// TwinCAT 3 PLC project SPS
// ProgramVersion: 3.1.4024.0
// libraries:
//   Tc2_MC2, * (Beckhoff Automation GmbH)
//   Tc2_Standard, * (Beckhoff Automation GmbH)
//   Tc2_System, * (Beckhoff Automation GmbH)
//   Tc3_Module, * (Beckhoff Automation GmbH)
// project tree:
//   DUTs/ eBetriebszustand.TcDUT
//   GVLs/ GVL_PosKinematic.TcGVL, IFC_HW.TcGVL (not stored)
//   / PlcTask.TcTTO
//   POUs/ FB_Abfuellmodul.TcPOU, FB_Ampel.TcPOU, FB_Blinklicht.TcPOU, FB_Dispenser.TcPOU, FB_EZylinder.TcPOU, FB_Manipulatormodul.TcPOU, FB_Maschinentuer.TcPOU, FB_TEST.TcPOU, FUN_SCALE.TcPOU, MAIN.TcPOU, FB_Vereinzelung.TcPOU
//   POUs/Manipulator/ FB_MANACHSE.TcPOU, FB_Robotsteuerung.TcPOU
//   POUs/Transport/ FB_Foerderband.TcPOU, FB_Transport.TcPOU, FB_TransportA.TcPOU, FB_TransportE.TcPOU, FB_TransportLogik.TcPOU
// real-time tasks:
//   TASK PlcTask: cycle T#10ms, priority 20, ADS port 350
// motion (NC):
//   TASK NC-Task 1 SAF: cycle T#2ms, priority 4, ADS port 501
//   TASK NC-Task 1 SVB: cycle T#10ms, priority 8, ADS port 511
//   AXIS Conveyer (id 1)
//     Dynamic: AccelerationMaximum=700, DecelerationMaximum=700, Acceleration=400, Deceleration=400, Jerk=6000
//     Velo: Maximum=50
//     OtherSettings: AllowMotionCmdToSlave=true
//     encoder EncType=1
//     drive DrvType=5
//       Analog: VeloReferenz=50, TorqueSetpointScale=10, ScaleFactorActTorque=0.1
//       TimeComp: TaskDelayCycles=1
//     controller CtrType=1
//       CtrPara: PriorControlFactor=1
//         Observer: BandWidth=20
//   AXIS Dispenser1 (id 2)
//     Dynamic: AccelerationMaximum=700, DecelerationMaximum=700, Acceleration=400, Deceleration=400, Jerk=6000
//     Velo: Maximum=50
//     OtherSettings: AllowMotionCmdToSlave=true
//     encoder EncType=1
//     drive DrvType=5
//       Analog: VeloReferenz=50, TorqueSetpointScale=10, ScaleFactorActTorque=0.1
//       TimeComp: TaskDelayCycles=1
//     controller CtrType=1
//       CtrPara: PriorControlFactor=1
//         Observer: BandWidth=20
//   AXIS Dispenser2 (id 3)
//     Dynamic: AccelerationMaximum=700, DecelerationMaximum=700, Acceleration=400, Deceleration=400, Jerk=6000
//     Velo: Maximum=50
//     OtherSettings: AllowMotionCmdToSlave=true
//     encoder EncType=1
//     drive DrvType=5
//       Analog: VeloReferenz=50, TorqueSetpointScale=10, ScaleFactorActTorque=0.1
//       TimeComp: TaskDelayCycles=1
//     controller CtrType=1
//       CtrPara: PriorControlFactor=1
//         Observer: BandWidth=20
//   AXIS Dispenser3 (id 4)
//     Dynamic: AccelerationMaximum=700, DecelerationMaximum=700, Acceleration=400, Deceleration=400, Jerk=6000
//     Velo: Maximum=50
//     OtherSettings: AllowMotionCmdToSlave=true
//     encoder EncType=1
//     drive DrvType=5
//       Analog: VeloReferenz=50, TorqueSetpointScale=10, ScaleFactorActTorque=0.1
//       TimeComp: TaskDelayCycles=1
//     controller CtrType=1
//       CtrPara: PriorControlFactor=1
//         Observer: BandWidth=20
//   AXIS ManAchseX (id 5)
//     Dynamic: AccelerationMaximum=700, DecelerationMaximum=700, Acceleration=400, Deceleration=400, Jerk=6000
//     Velo: Maximum=30
//     OtherSettings: AllowMotionCmdToSlave=true
//     encoder EncType=1
//       EncPara: ScaleFactorNumerator=0.0025
//         Inc: RefSearchInverse=true, RefSyncInverse=false
//     drive DrvType=5
//       Analog: VeloReferenz=30, TorqueSetpointScale=10, ScaleFactorActTorque=0.1
//       TimeComp: TaskDelayCycles=1
//     controller CtrType=1
//       CtrPara: PriorControlFactor=1
//         Observer: BandWidth=20
//   AXIS ManAchseY (id 6)
//     Dynamic: AccelerationMaximum=700, DecelerationMaximum=700, Acceleration=400, Deceleration=400, Jerk=6000
//     Velo: Maximum=30
//     OtherSettings: AllowMotionCmdToSlave=true
//     encoder EncType=1
//       EncPara: ScaleFactorNumerator=0.0025
//         Inc: RefSearchInverse=true, RefSyncInverse=false
//     drive DrvType=5
//       Analog: VeloReferenz=30, TorqueSetpointScale=10, ScaleFactorActTorque=0.1
//       TimeComp: TaskDelayCycles=1
//     controller CtrType=1
//       CtrPara: PriorControlFactor=1
//         Observer: BandWidth=20
//   AXIS ManAchseZ (id 7)
//     Dynamic: AccelerationMaximum=700, DecelerationMaximum=700, Acceleration=400, Deceleration=400, Jerk=6000
//     Velo: Maximum=30
//     OtherSettings: AllowMotionCmdToSlave=true
//     encoder EncType=1
//       EncPara: ScaleFactorNumerator=0.0025
//         Inc: RefSearchInverse=true, RefSyncInverse=false
//     drive DrvType=5
//       Analog: VeloReferenz=30, TorqueSetpointScale=10, ScaleFactorActTorque=0.1
//       TimeComp: TaskDelayCycles=1
//     controller CtrType=1
//       CtrPara: PriorControlFactor=1
//         Observer: BandWidth=20
//   AXIS ManAchseG (id 8)
//     Dynamic: AccelerationMaximum=700, DecelerationMaximum=700, Acceleration=400, Deceleration=400, Jerk=6000
//     Velo: Maximum=30
//     OtherSettings: AllowMotionCmdToSlave=true
//     encoder EncType=1
//       EncPara: ScaleFactorNumerator=0.0025
//     drive DrvType=5
//       Analog: VeloReferenz=30, TorqueSetpointScale=10, ScaleFactorActTorque=0.1
//     controller CtrType=1
//       CtrPara: PriorControlFactor=1
//         Observer: BandWidth=20
// variable links:
//   SPS/SPS Instance <-> NC-Task 1 SAF/Axes/Conveyer
//     PlcTask Inputs/IFC_HW.ax_BandMotor.NcToPlc <-> Outputs/ToPlc
//     PlcTask Outputs/IFC_HW.ax_BandMotor.PlcToNc <-> Inputs/FromPlc
//   SPS/SPS Instance <-> NC-Task 1 SAF/Axes/Dispenser1
//     PlcTask Inputs/IFC_HW.ax_Extruder1.NcToPlc <-> Outputs/ToPlc
//     PlcTask Outputs/IFC_HW.ax_Extruder1.PlcToNc <-> Inputs/FromPlc
//   SPS/SPS Instance <-> NC-Task 1 SAF/Axes/Dispenser2
//     PlcTask Inputs/IFC_HW.ax_Extruder2.NcToPlc <-> Outputs/ToPlc
//     PlcTask Outputs/IFC_HW.ax_Extruder2.PlcToNc <-> Inputs/FromPlc
//   SPS/SPS Instance <-> NC-Task 1 SAF/Axes/Dispenser3
//     PlcTask Inputs/IFC_HW.ax_Extruder3.NcToPlc <-> Outputs/ToPlc
//     PlcTask Outputs/IFC_HW.ax_Extruder3.PlcToNc <-> Inputs/FromPlc
//   SPS/SPS Instance <-> NC-Task 1 SAF/Axes/ManAchseG
//     PlcTask Inputs/IFC_HW.ax_ManG.NcToPlc <-> Outputs/ToPlc
//     PlcTask Outputs/IFC_HW.ax_ManG.PlcToNc <-> Inputs/FromPlc
//   SPS/SPS Instance <-> NC-Task 1 SAF/Axes/ManAchseX
//     PlcTask Inputs/IFC_HW.ax_ManX.NcToPlc <-> Outputs/ToPlc
//     PlcTask Outputs/IFC_HW.ax_ManX.PlcToNc <-> Inputs/FromPlc
//   SPS/SPS Instance <-> NC-Task 1 SAF/Axes/ManAchseY
//     PlcTask Inputs/IFC_HW.ax_ManY.NcToPlc <-> Outputs/ToPlc
//     PlcTask Outputs/IFC_HW.ax_ManY.PlcToNc <-> Inputs/FromPlc
//   SPS/SPS Instance <-> NC-Task 1 SAF/Axes/ManAchseZ
//     PlcTask Inputs/IFC_HW.ax_ManZ.NcToPlc <-> Outputs/ToPlc
//     PlcTask Outputs/IFC_HW.ax_ManZ.PlcToNc <-> Inputs/FromPlc

CONFIGURATION SPS
    RESOURCE PLC ON TwinCAT3
        TASK PlcTask(INTERVAL := T#10ms, PRIORITY := 20);
        PROGRAM MAIN WITH PlcTask : MAIN;
    END_RESOURCE
END_CONFIGURATION

// ---- DUTs/eBetriebszustand.TcDUT
{attribute 'qualified_only'}
{attribute 'strict'}
TYPE eBetriebszustand :
(
	off, //nicht Betriebsbereit 
	error, //Fehlerbehafteter Stop(Sicherheitssteuerung)
	setup, //Wartung 
	warning, // Nicht fehlerbehafteter geplanter Stop 
	init, //Herstellung Betriebsbereitschaft 
	ready, //betriebsbereit 
	production, //Im Betrieb
	done, //Betrieb abgschlossen
	stop //geplanter Stillstand 
);
END_TYPE

// ---- GVLs/GVL_PosKinematic.TcGVL
{attribute 'qualified_only'}
VAR_GLOBAL
	// Home position
	pXhome : REAL := 29;
	pYhome : REAL := 145.5;
	pZhome : REAL := 45;
	
	// Conveyor position
	pXconv : REAL := 29;
	pYconv : REAL := 145.5;
	pZconv : REAL := 130;
	
	//Scale position
	pXscale : REAL := 36;
	pYscale : REAL := 7.5;
	pZscale : REAL := 131.5;
	
	// Heating position
	pXheat : REAL := 218.5;
	pYheat : REAL := 7;
	pZheat : REAL := 159;
	
	// Storage position
	pX1stor : REAL := 107;
	pX2stor : REAL := 158.7;
	pX3stor : REAL := 209.3;
	pX4stor : REAL := 260.3;
	pYstor : REAL := 139;
	pZstor : REAL := 120;
	
	// Z offset height
	pZoff : REAL := 45;
END_VAR

// ---- POUs/MAIN.TcPOU
PROGRAM MAIN
VAR
	fbBlinklicht : FB_Blinklicht;
	fbVereinzelung : FB_Vereinzelung;
	fbezylinder1 : FB_EZylinder;
	fbezylinder2 : FB_EZylinder;
	fbAmpel : FB_Ampel;
	fbTransport : FB_Transport;
	fbDispenser : FB_Dispenser;
	fbAbfuellmodul : FB_Abfuellmodul;
	fbManAchseX : FB_ManAchse;
	fbManAchseY : FB_ManAchse;
	fbManAchseZ : FB_ManAchse;
	fbManAchseG : FB_ManAchse;
	fbRobotsteuerung : FB_Robotsteuerung;
	fbManipulatormodul : FB_Manipulatormodul;
	ix : UINT;
	ry : REAL;
	ax : Axis_Ref;
END_VAR

ry := FUN_SCALE(TO_REAL(ix),4096,0,350,0);

	
fbAbfuellmodul(
	bEnable:= IFC_HW.bEnable, 
	bExecute:= IFC_HW.bExecute, 
	nstation:= , 
	bEinzelSens1:= IFC_HW.bEinzelSens1, 
	bEinzelSens2:= IFC_HW.bEinzelSens2, 
	bEinzelSens3:= IFC_HW.bEinzelSens3, 
	bEinzelSens4:= IFC_HW.bBandSens1, 
	bBandSens1:= IFC_HW.bBandSens1, 
	bBandSens2:= IFC_HW.bBandSens2, 
	bBandSens3:= IFC_HW.bBandSens3, 
	bBandSens4:= IFC_HW.bBandSens4, 
	bstopper1=> IFC_HW.bBandHub1, 
	bstopper2=> IFC_HW.bBandHub2, 
	bstopper3=>IFC_HW.bBandHub3, 
	estate=> , 
	bgate1=> fbeZylinder1.bgate, 
	bgate2=> fbeZylinder2.bgate, 
	axTransport:= IFC_HW.ax_BandMotor, 
	axDisp1:= IFC_HW.ax_Extruder1, 
	axDisp2:= IFC_HW.ax_Extruder2, 
	axDisp3:= IFC_HW.ax_Extruder3);
	
	fbezylinder1(bgate:= , berror:= , bR1=>IFC_HW.bR1AKT1 , bR2=>IFC_HW.br2AKT1 );
	
	fbezylinder2(bgate:= , berror:= , bR1=>IFC_HW.bR1AKT2 , bR2=> IFC_HW.bR2AKT2);
	
	
	fbAmpel(estate:= fbAbfuellmodul.estate, bAmpelgruen=>IFC_HW.bAmpelGrun , bAmpelrot=>IFC_HW.bAmpelRot , bAmpelgelb=>IFC_HW.bAmpelGelb );

fbManipulatormodul(
	bEnable:= IFC_Hw.bEnable, 
	bExecute:= IFC_Hw.bExecute, 
	pXhome:= GVL_PosKinematic.pXhome, 
	pYhome:= GVL_PosKinematic.pYhome, 
	pZhome:= GVL_PosKinematic.pZhome, 
	pXconv:= GVL_PosKinematic.pXconv, 
	pYconv:= GVL_PosKinematic.pYconv, 
	pZconv:= GVL_PosKinematic.pZconv, 
	pXscale:= GVL_PosKinematic.pXscale, 
	pYscale:= GVL_PosKinematic.pYscale, 
	pZscale:= GVL_PosKinematic.pZscale, 
	pXheat:= GVL_PosKinematic.pXheat, 
	pYheat:= GVL_PosKinematic.pYheat, 
	pZheat:= GVL_PosKinematic.pZheat, 
	pX1stor:= GVL_PosKinematic.pX1stor, 
	pX2stor:= GVL_PosKinematic.pX2stor, 
	pX3stor:= GVL_PosKinematic.pX3stor, 
	pX4stor:= GVL_PosKinematic.pX4stor, 
	pYstor:= GVL_PosKinematic.pYstor, 
	pZstor:= GVL_PosKinematic.pZstor, 
	estateE:= fbAbfuellmodul.estate, 
	bxEndschalter:= IFC_HW.bManEndXmin, 
	byEndschalter:= IFC_HW.bManEndYmin, 
	bzEndschalter:= IFC_HW.bManEndZmin, 
	bGEndschalter:= IFC_HW.bManEndGmin, 
	estate=> , 
	ax_ManX:= IFC_HW.ax_ManX, 
	ax_ManY:= IFC_HW.ax_ManY, 
	ax_ManZ:= IFC_HW.ax_ManZ, 
	ax_ManG:= IFC_HW.ax_ManG);

(*
fbRobotsteuerung(
	bEnable:= IFC_Hw.bEnable, 
	bExecute:= IFC_Hw.bExecute, 
	bxposition:= GVL_PosKinematic.pXconv, 
	byposition:= GVL_PosKinematic.pYconv, 
	bzposition:= GVL_PosKinematic.pZconv, 
	bxEndschalter:= IFC_HW.bManEndXmin, 
	byEndschalter:= IFC_HW.bManEndYmin, 
	bzEndschalter:= IFC_HW.bManEndZmin, 
	bGEndschalter:= IFC_HW.bManEndGmin, 
	estateE:= fbAbfuellmodul.estate, 
	estate=> , 
	movedone=> , 
	ax_ManX:= IFC_HW.ax_ManX, 
	ax_ManY:= IFC_HW.ax_ManY, 
	ax_ManZ:= IFC_HW.ax_ManZ, 
	ax_ManG:= IFC_HW.ax_ManG);

fbManAchseX(
	benable:= IFC_Hw.bEnable, 
	bexecute:= IFC_Hw.bExecute, 
	bEndschalter:= IFC_HW.bManEndXmin, 
	rPosition:= GVL_PosKinematic.pXconv, 
	rVel:= 30, 
	estate=> , 
	ax:= IFC_HW.ax_ManX);
	
fbManAchseY(
	benable:= IFC_Hw.bEnable, 
	bexecute:= IFC_Hw.bExecute, 
	bEndschalter:= IFC_HW.bManEndYmin, 
	rPosition:= GVL_PosKinematic.pYconv, 
	rVel:= 30, 
	estate=> , 
	ax:= IFC_HW.ax_ManY); 

fbManAchseZ(
	benable:= IFC_Hw.bEnable, 
	bexecute:= IFC_Hw.bExecute, 
	bEndschalter:= IFC_HW.bManEndZmin, 
	rPosition:= GVL_PosKinematic.pZconv, 
	rVel:= 30, 
	estate=> , 
	ax:= IFC_HW.ax_ManZ); 	

fbManAchseG(
	benable:= IFC_Hw.bEnable, 
	bexecute:= IFC_Hw.bExecute, 
	bEndschalter:= IFC_HW.bManEndGmin, 
	rPosition:= 2, 
	rVel:= 30, 
	estate=> , 
	ax:= IFC_HW.ax_ManG);
*)

END_PROGRAM

// ---- POUs/FB_Blinklicht.TcPOU
FUNCTION_BLOCK FB_Blinklicht
VAR_INPUT
	bStartStop	: BOOL;
	tPeriode	: TIME := T#1.5S;
END_VAR
VAR_OUTPUT
	bBlink	:BOOL;
END_VAR
VAR
	fbTon	:Ton;
	fbRtrig	:R_Trig;
	bEinAus	:BOOL;
END_VAR

fbRtrig(CLK:= bStartStop , Q=> );

IF fbRtrig.Q THEN
	bEinAus := NOT bEinAus;
END_IF

//fbTon.IN := bBlink AND NOT fbTon.Q;
//fbTon.PT := T#1S;

fbTon(IN:=bEinAus AND NOT fbTon.Q , PT:=T#1.5S , Q=> , ET=> );


IF fbTon.ET <= fbTon.PT/2 THEN 
	bBlink := FALSE;
ELSIF fbTon.ET > fbTon.PT/2 THEN
	bBlink := TRUE;
END_IF

END_FUNCTION_BLOCK

// ---- POUs/FB_Vereinzelung.TcPOU
FUNCTION_BLOCK FB_Vereinzelung 
VAR_INPUT
	//Steuervariablen
	benable : BOOL;
	bexecute : BOOL;
	// Hardware Eingänge
	bsensor1 : BOOL; //Flasche in der Kammer 
	bsensor2 : BOOL; //Flasche inm Rohr 
	bsensor3 : BOOL; //Flasche auf Kopf
	bsensor4 : BOOL; //Flasche am Förderband
	
END_VAR
VAR_OUTPUT
	//Hardwareausgänge 
	bgate1 : BOOL;
	bgate2 : BOOL;
	//Steuervariable 
	estate : eBetriebszustand;
END_VAR
VAR
	nstate : INT := 100;
	fbTon : Ton;
END_VAR

fbTon(IN:= , PT:=T#1S , Q=> , ET=> );

CASE nstate OF 
	100:
	eState :=eBetriebszustand.off;
	
	IF bsensor1 AND benable THEN 
		nstate := 21;//Ready
	ELSIF benable THEN
		nstate := 0; //Init		
	END_IF
	
	0: // Kammer ist leer 
	estate := eBetriebszustand.init;
	bgate1 := FALSE;
	bgate2 := FALSE;
	
	IF bsensor2 AND NOT bsensor3 THEN
		nstate := 1; //Schleuße Oben öffnen
	END_IF
	
	1: // Schleuße oben öffnen
	estate := eBetriebszustand.init;
	bgate1 := TRUE;
	bgate2 := FALSE;
	
	IF bsensor1 THEN
		nstate := 2; //Schleuße oben schließen
	END_IF
	
	2: //Schleuße oben schließen
	estate := eBetriebszustand.init;
	bgate1 := FALSE;
	bgate2 := FALSE;
	fbTon.In := TRUE;
	
	IF fbTon.Q THEN
		nstate := 21; //ready
		fbTon.IN := FALSE;
	END_IF
	
	21: //ready
	estate:= eBetriebszustand.ready;
	bgate1:= FALSE;
	bgate2:= FALSE;
	
	
	IF bexecute THEN
		nstate := 3; //Schleuße unten öffnen
	END_IF
	
	3: //Schleuße unten öffnen
	estate:= eBetriebszustand.production;
	bgate1:= FALSE;
	bgate2:= TRUE;
	
	IF bsensor4 THEN
		nstate := 4; //Schleuße unten schließen
	END_IF
	
	4: //Schleuße unten schließen
	estate:= eBetriebszustand.production;
	bgate1:= FALSE;
	bgate2:= FALSE;
	fbTon.IN:= TRUE;
	
	IF fbTon.Q THEN
		nstate := 41; //done
		fbTon.IN := FALSE;
	END_IF	
	
	41: //Done
	estate:= eBetriebszustand.done;
	bgate1:= FALSE;
	bgate2:= FALSE;
	
	IF NOT bexecute THEN
		nstate:= 0; //Kammer leer
	END_IF
	
END_CASE

END_FUNCTION_BLOCK

// ---- POUs/FB_EZylinder.TcPOU
FUNCTION_BLOCK FB_EZylinder
VAR_INPUT
	bgate : BOOL;
	berror : BOOL;
END_VAR
VAR_OUTPUT
	bR1 : BOOL;
	bR2 : BOOL;
END_VAR
VAR
END_VAR


bR1 := bgate;
bR2 := NOT bgate;

IF berror THEN
	bR1 := FALSE;
	bR2 := FALSE;
	
END_IF

END_FUNCTION_BLOCK

// ---- POUs/FB_Ampel.TcPOU
FUNCTION_BLOCK FB_Ampel
VAR_INPUT
	estate : eBetriebszustand;
END_VAR
VAR_OUTPUT
	bAmpelgruen : BOOL;
	bAmpelrot : BOOL;
	bAmpelgelb : BOOL;
END_VAR
VAR
	Ampel_blinken : FB_Blinklicht;
END_VAR

//Die Ampel leuchtet je nach Betriebszustand in unterschiedlichen Farben, um diesen anzuzeigen
CASE estate OF
	
	eBetriebszustand.off:
	bAmpelgruen := FALSE;
	bAmpelrot := TRUE;
	bAmpelgelb := FALSE;	
	
	eBetriebszustand.init:
	bAmpelrot := FALSE;
	bAmpelgelb := FALSE;
	Ampel_blinken(bStartStop:=TRUE , tPeriode:= , bBlink=>bAmpelgruen );
	
	eBetriebszustand.ready:
	bAmpelrot := FALSE;
	Ampel_blinken(bStartStop:=TRUE , tPeriode:= , bBlink=>bAmpelgelb );
	bAmpelgruen := NOT bAmpelgelb;
	//gruen_blinken(bStartStop:=True , tPeriode:= , bBlink=>bAmpelgruen );
	
	eBetriebszustand.production:
	bAmpelrot := FALSE;
	bAmpelgelb := FALSE;
	bAmpelgruen := TRUE;
	
	eBetriebszustand.done:
	bAmpelgruen := TRUE;
	bAmpelrot := FALSE;
	bAmpelgelb := TRUE;	
	
END_CASE

END_FUNCTION_BLOCK

// ---- POUs/Transport/FB_Transport.TcPOU
FUNCTION_BLOCK FB_Transport
VAR_INPUT
	bEnable : BOOL;
	bExecute : BOOL;
	nstation : INT;
	//Hardware Eingänge
	bSens1 : BOOL;
	bSens2 : BOOL;
	bSens3 : BOOL;
	bSens4 : BOOL;
END_VAR
VAR_OUTPUT
	eState : eBetriebszustand;
	bstopper1 : BOOL;
	bstopper2 : BOOL;
	bstopper3 : BOOL;
	
END_VAR
VAR
	fbTransportE : FB_TransportE;
	fbTransportLogik : FB_TransportLogik;
	fbTransportBand : FB_Foerderband;
	fbTransportA : FB_TransportA;
END_VAR
VAR_IN_OUT
	//Achsenreferenz
	ax : Axis_Ref;
END_VAR

fbTransportE(
	bSens1:= bSens1, 
	bSens2:= bSens2, 
	bSens3:= bSens3, 
	bSens4:= bSens4, 
	bStation1=> , 
	bStation2=> , 
	bStation3=> , 
	bStation4=> );
	
	
fbTransportLogik(
	bEnable:= bEnable, 
	bExecute:= bExecute, 
	eStateE:= fbTransportBand.estate, 
	nStation:= nstation, 
	bStation1:= fbTransportE.bStation1, 
	bStation2:= fbTransportE.bStation2, 
	bStation3:= fbTransportE.bStation3, 
	bStation4:= fbTransportE.bStation4, 
	bEnableA=> , 
	bExecuteA=> , 
	bStopA=> , 
	eStateA=> estate, 
	bStop1=> , 
	bStop2=> , 
	bStop3=> );	
	
fbTransportBand(
	benable:= fbTransportLogik.bEnableA, 
	bexecute:= fbTransportLogik.bExecuteA, 
	bhalt:= fbTransportLogik.bStopA, 
	rVel:= 30, 
	eDirection:= MC_Positive_Direction, 
	estate=> , 
	ax:= ax);

fbTransportA(
	bstop1:= fbTransportLogik.bStop1, 
	bstop2:= fbTransportLogik.bStop2, 
	bstop3:= fbTransportLogik.bStop3, 
	bstopper1=> bStopper1, 
	bstopper2=> bStopper2, 
	bstopper3=> bStopper3);

END_FUNCTION_BLOCK

// ---- POUs/Transport/FB_TransportE.TcPOU
FUNCTION_BLOCK FB_TransportE
VAR_INPUT
	bSens1 : BOOL;
	bSens2 : BOOL;
	bSens3 : BOOL;
	bSens4 : BOOL;
END_VAR
VAR_OUTPUT
	bStation1 : BOOL;
	bStation2 : BOOL;
	bStation3 : BOOL;
	bStation4 : BOOL;
END_VAR
VAR
END_VAR

bStation1 := bSens1;
bStation2 := bSens2;
bStation3 := bSens3;
bStation4 := bSens4;

END_FUNCTION_BLOCK

// ---- POUs/Transport/FB_TransportLogik.TcPOU
FUNCTION_BLOCK FB_TransportLogik
VAR_INPUT
	bEnable : BOOL;
    bExecute : BOOL;
    eStateE : eBetriebszustand;
    nStation : INT := 0;

    // Logiksignale -> Hardware Signale
    bStation1 : BOOL;
    bStation2 : BOOL;
    bStation3 : BOOL;
    bStation4 : BOOL;
END_VAR
VAR_OUTPUT
	bEnableA : BOOL;
    bExecuteA : BOOL;
    eStateA : eBetriebszustand;
	bStopA : BOOL;
    //Hardware Signale -> Logik
    bStop1 : BOOL;
    bStop2 : BOOL;
    bStop3 : BOOL;
END_VAR
VAR
	nstate : INT;
END_VAR

CASE nstate OF 
	0: //Off
	bEnableA := FALSE;
	bExecuteA := FALSE;
	bStopA := FALSE;
	bStop1 := FALSE;
	bStop2 := FALSE;
	bStop3 := FALSE;
	eStateA    := eBetriebszustand.off;
	
	IF bEnable THEN
		nstate := 1; //Init
	END_IF
	
	1: //Init
	bEnableA := TRUE;
	bExecuteA := FALSE;
	bStopA := FALSE;
	bStop1 := FALSE;
	bStop2 := FALSE;
	bStop3 := FALSE;
	eStateA    := eBetriebszustand.init;

	IF eStateE = eBetriebszustand.ready THEN
		nstate := 2; //Ready
	END_IF

	2: //Ready
	bEnableA := TRUE;
	bExecuteA := FALSE;
	bStopA := FALSE;
	bStop1 := FALSE;
	bStop2 := FALSE;
	bStop3 := FALSE;
	eStateA    := eBetriebszustand.ready;
	
	IF bExecute THEN
		nstate := 3; //Förderband Start
	END_IF
	
	3: //Förderband Start
	
	bExecuteA := TRUE;
	eStateA    := eBetriebszustand.production;
	
	IF (nStation -1) = 1 THEN
		bStop1 := TRUE;
	ELSIF (nStation - 1) = 2 THEN
		bStop2 := TRUE;
	ELSIF (nStation - 1) = 3 THEN
		bStop3 := TRUE;
	END_IF
	
	IF bStation1 AND (nStation = 1) THEN
		nstate := 4; //Förderband Stop
	ELSIF bStation2 AND (nStation = 2) THEN
		nstate := 4; //Förderband Stop
	ELSIF bStation3 AND (nStation = 3) THEN
		nstate := 4; //Förderband Stop
	ELSIF bStation4 AND (nStation = 4) THEN
		nstate := 4; //Förderband Stop
	END_IF
	
	4: // Förderband Stop
	bExecuteA := FALSE;
	bStopA := TRUE;
	
	IF (nStation -1) = 1 THEN
		bStop1 := FALSE;
	ELSIF (nStation - 1) = 2 THEN
		bStop2 := FALSE;
	ELSIF (nStation - 1) = 3 THEN
		bStop3 := FALSE;
	END_IF
	
	IF estateE = eBetriebszustand.done THEN
		nstate := 5; // Done
	END_IF
	
	5: // Done
	eStateA    := eBetriebszustand.done;
	
	IF NOT bExecute THEN
		nstate := 2; // Ready
	END_IF
	
END_CASE

END_FUNCTION_BLOCK

// ---- POUs/Transport/FB_Foerderband.TcPOU
FUNCTION_BLOCK FB_Foerderband
VAR_INPUT
	//Steuereingänge
	benable : BOOL;
	bexecute : BOOL;
	bhalt : BOOL;
	rVel : INT := 30; //mm per s
	
	eDirection : MC_Direction := MC_Positive_Direction;
END_VAR
VAR_OUTPUT
	estate: eBetriebszustand;
END_VAR
VAR
	nstate : INT := 0;
	
	//Motion Blöcke der Tc2_Mc2
	mcReset : MC_Reset;
	mcPower : MC_Power;
	mcMove : MC_MoveVelocity;
	mcHalt : MC_Halt;
	
	bAxPower : BOOL;
	bAXMove : BOOL;
	
	fbTon	:Ton;
END_VAR
VAR_IN_OUT
	ax : AXIS_REF;
END_VAR

// update our axis
ax.ReadStatus();

mcReset(Axis := ax); 

mcPower(
	Axis:= ax, 
	Enable:= bAxPower, 
	Enable_Positive:= bAxPower, 
	Enable_Negative:= bAxPower, 
	Override:= 100);

mcMove(
	Axis:= ax, 
	Execute:= bAxMove , 
	Velocity:= rVel,
	Acceleration:= 60.0, 
	Direction:= eDirection);
	
mcHalt(
	Axis:= ax, 
	Execute:= ,
	Deceleration:= 60.0);
	
fbTon(
  IN := bhalt,   
  PT := T#1S
);
	
(*
IF NOT benable THEN
	nstate := 0;
END_IF
*)

CASE nstate OF 
	
	0: //off
	estate := eBetriebszustand.off;
	bAxPower := FALSE;
	bAxMove := FALSE;
	
	IF McPower.Status AND benable THEN
		nstate := 20; //Ready
	END_IF
	IF NOT McPower.Status AND bEnable THEN
		nstate:=10;
	END_IF
	
	10: // INIT_Reset
	estate := eBetriebszustand.init;
	mcReset.Execute := TRUE;
	bAxPower:= FALSE;
	bAxMove:= FALSE;
	bhalt:= False;
	
	IF McReset.Done THEN
		nstate:= 11; //INIT-Power
	END_IF
	
	11: //INIT-Power
	estate := eBetriebszustand.init;
	bAxPower := TRUE;
	
	IF Mcpower.Status THEN
		nstate := 20; //Ready
	END_IF
	
	20: //Ready
	estate:= eBetriebszustand.ready;
	mcHalt.Execute := FALSE;
	bAxMove := FALSE;
	
	IF bexecute THEN
		nstate := 30; // Move
	END_IF
	
	30: //Move
	estate := eBetriebszustand.production;
	bAxMove := TRUE;

	IF bhalt THEN
		nstate := 31; //Warten
	END_IF
	
	31: //Warten
	estate := eBetriebszustand.production;
	bAxMove := TRUE;
	
	IF fbTOn.Q THEN
		nstate:= 32; //Halten
	END_IF
	
	32: //Halten
	estate := eBetriebszustand.production;
    mcHalt.Execute := TRUE;
	
	IF mchalt.Done THEN
		nstate := 40; //Fertig
	END_IF
	40: //Fertig
	estate := eBetriebszustand.done;
	mcHalt.Execute := FALSE;
	
	IF NOT bexecute THEN
		nstate := 20; // Ready
	END_IF
	
END_CASE

END_FUNCTION_BLOCK

// ---- POUs/Transport/FB_TransportA.TcPOU
FUNCTION_BLOCK FB_TransportA
VAR_INPUT
	bstop1 : BOOL;
	bstop2 : BOOL;
	bstop3 : BOOL;
END_VAR
VAR_OUTPUT
	//Hardware Signale
	bstopper1 : BOOL;
	bstopper2 : BOOL;
	bstopper3 : BOOL;
END_VAR
VAR
END_VAR

bstopper1 := bstop1;
bstopper2 := bstop2;
bstopper3 := bstop3;

END_FUNCTION_BLOCK

// ---- POUs/FB_Dispenser.TcPOU
FUNCTION_BLOCK FB_Dispenser
VAR_INPUT
	//Steuereingänge
	benable : BOOL;
	bexecute : BOOL;
	rVelocity : INT;
	rDistance : INT; 
	
END_VAR
VAR_OUTPUT
	estate: eBetriebszustand;
END_VAR
VAR
	nstate : INT := 0;
	
	//Motion Blöcke der Tc2_Mc2
	mcReset : MC_Reset;
	mcPower : MC_Power;
	mcMove : MC_MoveRelative;
	
	bAxPower : BOOL;
	bAXMove : BOOL;
	
END_VAR
VAR_IN_OUT
	ax : AXIS_REF;
END_VAR

// update our axis
ax.ReadStatus();

mcReset(Axis := ax); 

mcPower(
	Axis:= ax, 
	Enable:= bAxPower, 
	Enable_Positive:= bAxPower, 
	Enable_Negative:= bAxPower, 
	Override:= 100);

mcMove(
	Axis:= ax, 
	Execute:= bAxMove, 
	Distance:= rDistance, 
	Velocity:= rVelocity, 
	Acceleration:= 60.0, 
	Deceleration:= 60.0);

	

IF NOT benable THEN
	nstate := 0;
END_IF

CASE nstate OF 
	
	0: //off
	estate := eBetriebszustand.off;
	bAxPower := FALSE;
	bAxMove := FALSE;
	
	IF McPower.Status AND benable THEN
		nstate := 20; //Ready
	END_IF
	IF NOT McPower.Status AND bEnable THEN
		nstate:=10;
	END_IF
	
	10: // INIT_Reset
	estate := eBetriebszustand.init;
	mcReset.Execute := TRUE;
	bAxPower:= FALSE;
	bAxMove:= FALSE;
	
	IF McReset.Done THEN
		nstate:= 11; //INIT-Power
	END_IF
	
	11: //INIT-Power
	estate := eBetriebszustand.init;
	bAxPower := TRUE;
	
	IF Mcpower.Status THEN
		nstate := 20; //Ready
	END_IF
	
	20: //Ready
	estate:= eBetriebszustand.ready;
	bAxMove := FALSE;
	
	IF bexecute THEN
		nstate := 30; // Move
	END_IF
	
	30: //Move
	estate := eBetriebszustand.production;
	bAxMove := TRUE;

	IF mcmove.Done THEN
		nstate := 40; //Done
	END_IF
	
	40: //Done
	estate := eBetriebszustand.done;
	
	
	IF NOT bexecute THEN
		nstate := 20; // Ready
	END_IF
	
END_CASE

END_FUNCTION_BLOCK

// ---- POUs/FB_Abfuellmodul.TcPOU
FUNCTION_BLOCK FB_Abfuellmodul
VAR_INPUT
	bEnable : BOOL;
	bExecute : BOOL;
	
    // Vereinzelungs-Sensoren
    bEinzelSens1 : BOOL;
    bEinzelSens2 : BOOL;
    bEinzelSens3 : BOOL;
    bEinzelSens4 : BOOL;
 		
	// Foerderband-Sensoren
	bBandSens1 : BOOL;
	bBandSens2 : BOOL;
	bBandSens3 : BOOL;
	bBandSens4 : BOOL;
	
	
END_VAR
VAR_OUTPUT
	estate : eBetriebszustand;
	bgate1 : BOOL;
	bgate2 : BOOL;
	
	bstopper1 : BOOL;
	bstopper2 : BOOL;
	bstopper3 : BOOL;
END_VAR
VAR
	fbVereinzelung : FB_Vereinzelung;
	fbTransport : FB_Transport;
	fbDispenser1 : FB_Dispenser;
	fbDispenser2 : FB_Dispenser;
	fbDispenser3 : FB_Dispenser;
	nstate : INT := 0;
	nStation : INT;
	Vcounter : INT;
END_VAR
VAR_IN_OUT
    // Achsen-Referenzen 
    axTransport: AXIS_REF;   // Foerderband‐Achse
    axDisp1    : AXIS_REF;   // Dispenser 1
    axDisp2    : AXIS_REF;   // Dispenser 2
    axDisp3    : AXIS_REF;   // Dispenser 3
END_VAR

fbVereinzelung(
	benable:= , 
	bexecute:= , 
	bsensor1:= bEinzelSens1, 
	bsensor2:= bEinzelSens2, 
	bsensor3:= bEinzelSens3, 
	bsensor4:= bEinzelSens4, 
	bgate1=> bgate1, 
	bgate2=> bgate2, 
	estate=> );

fbTransport(
	bEnable:= , 
	bExecute:= , 
	nstation:= nstation, 
	bSens1:= bBandSens1, 
	bSens2:= bBandSens2, 
	bSens3:= bBandSens3, 
	bSens4:= bBandSens4, 
	eState=> , 
	bstopper1=> bstopper1, 
	bstopper2=> bstopper2, 
	bstopper3=> bstopper3, 
	ax:= axTransport);
	
fbDispenser1(
	benable:= , 
	bexecute:= , 
	rVelocity:= 10, 
	rDistance:= 10, 
	estate=> , 
	ax:= axDisp1);
	
fbDispenser2(
	benable:= , 
	bexecute:= , 
	rVelocity:= 10, 
	rDistance:= 10, 
	estate=> , 
	ax:= axDisp2);
	
fbDispenser3(
	benable:= , 
	bexecute:= , 
	rVelocity:= 10, 
	rDistance:= 10, 
	estate=> , 
	ax:= axDisp3);
	

CASE nstate OF 
	0: // Off
	fbVereinzelung.benable := FALSE;
	fbTransport.bEnable := FALSE;
	fbDispenser1.bEnable := FALSE;
	fbDispenser2.bEnable := FALSE;
	fbDispenser3.bEnable := FALSE;
	
	
	fbVereinzelung.bexecute := FALSE;
	fbTransport.bExecute := FALSE;
	fbDispenser1.bExecute := FALSE;
	fbDispenser2.bExecute := FALSE;
	fbDispenser3.bExecute := FALSE;
	
	eState :=eBetriebszustand.off;
	
	IF bEnable THEN
		nstate := 10; // Init
	END_IF
	
	10: // Init
	fbVereinzelung.benable := TRUE;
	fbTransport.bEnable := TRUE;
	fbDispenser1.bEnable := TRUE;
	fbDispenser2.bEnable := TRUE;
	fbDispenser3.bEnable := TRUE;
	
	
	fbVereinzelung.bexecute := FALSE;
	fbTransport.bExecute := FALSE;
	fbDispenser1.bExecute := FALSE;
	fbDispenser2.bExecute := FALSE;
	fbDispenser3.bExecute := FALSE;
	
	eState :=eBetriebszustand.init;
	
	IF fbVereinzelung.estate = eBetriebszustand.ready AND 
		fbTransport.estate = eBetriebszustand.ready AND
		fbDispenser1.estate = eBetriebszustand.ready AND
		fbDispenser2.estate = eBetriebszustand.ready AND
		fbDispenser3.estate = eBetriebszustand.ready THEN
		
		nstate := 20; // Ready
	END_IF
	
	20: // Ready
	fbVereinzelung.benable := TRUE;
	fbTransport.bEnable := TRUE;
	fbDispenser1.bEnable := TRUE;
	fbDispenser2.bEnable := TRUE;
	fbDispenser3.bEnable := TRUE;
	nstation := 1;
	
	estate := eBetriebszustand.ready;
	IF bExecute THEN
		nState := 30; //Move
	END_IF
	
	
	30: // Move
	eState := eBetriebszustand.Production;
	fbVereinzelung.benable := FALSE;
	fbTransport.bEnable := TRUE;
	fbDispenser1.bEnable := TRUE;
	fbDispenser2.bEnable := TRUE;
	fbDispenser3.bEnable := TRUE;
	
	fbVereinzelung.bExecute := FALSE;
	fbDispenser1.bExecute := FALSE;
	fbDispenser2.bExecute := FALSE;
	fbDispenser3.bExecute := FALSE;
	
	CASE nstation OF 
		1:
		fbVereinzelung.benable  := TRUE;
		fbVereinzelung.bexecute := TRUE;
		fbTransport.bExecute := TRUE;
		IF FbTransport.eState = eBetriebszustand.done AND 
			FbVereinzelung.estate = ebetriebszustand.done AND
			bBandsens1 THEN
			fbVereinzelung.benable  := FALSE;
			fbVereinzelung.bexecute := FALSE;
			FbTransport.bExecute := FALSE;
			nState := 40;
		END_IF
		2:
		fbTransport.bExecute := TRUE;
		IF FbTransport.eState = eBetriebszustand.done AND bBandsens2 THEN
			FbTransport.bExecute := FALSE;
			nstate:=40;
		END_IF
		3:
		fbTransport.bExecute := TRUE;
		IF FbTransport.eState = eBetriebszustand.done AND bBandsens3 THEN
			FbTransport.bExecute := FALSE;
			nstate:=40;
		END_IF
		4:
		fbTransport.bExecute := TRUE;
		IF FbTransport.eState = eBetriebszustand.done AND bBandsens4 THEN
			FbTransport.bExecute := FALSE;
			nstate:=50;
		END_IF
		END_CASE
		

	40: //Bottling
	eState := eBetriebszustand.production;
	
    CASE nStation OF
      1: 
	  fbDispenser1.bExecute := TRUE;
	  IF (nStation =1 AND fbDispenser1.eState=eBetriebszustand.done) THEN
		  FbDispenser1.bExecute := FALSE;
		  nStation := 2;
		  nState := 30;
	  END_IF
	  
      2: 
	  fbDispenser2.bExecute := TRUE;
	  IF (nStation =2 AND fbDispenser2.eState=eBetriebszustand.done) THEN
		  FbDispenser2.bExecute := FALSE;
		  nStation := 3;
		  nState := 30;
	  END_IF
	  3:
	  fbDispenser3.bExecute := TRUE;
	  IF (nStation =3 AND fbDispenser3.eState=eBetriebszustand.done) THEN
		  FbDispenser3.bExecute := FALSE;
		  nStation := 4;
		  nState := 30;
	  END_IF
    END_CASE
	
	
	50: // Done
	
	estate:= eBetriebszustand.done;
	
	fbTransport.bExecute := FALSE;
	fbDispenser1.bExecute := FALSE;
	fbDispenser2.bExecute := FALSE;
	fbDispenser3.bExecute := FALSE;
	
	
	
END_CASE

END_FUNCTION_BLOCK

// ---- POUs/Manipulator/FB_MANACHSE.TcPOU
FUNCTION_BLOCK FB_MANACHSE
VAR_INPUT
	//Steuereingänge
	benable : BOOL;
	bexecute : BOOL;
	bEndschalter : BOOL;
	rPosition     : LREAL := 0.0;
	rVel : INT := 30; //mm per s
	
END_VAR
VAR_OUTPUT
	estate: eBetriebszustand;
END_VAR
VAR
	nstate : INT := 0;
	
	//Motion Blöcke der Tc2_Mc2
	mcReset : MC_Reset;
	mcPower : MC_Power;
	mcHome : MC_HOME;
	mcMove : MC_MoveAbsolute;

	// interne Flags
	bAxPower : BOOL;
	bAXMove : BOOL;
    homeDone      : BOOL;
    moveDone      : BOOL;	

	
END_VAR
VAR_IN_OUT
	ax : AXIS_REF;
END_VAR

// update our axis
ax.ReadStatus();

mcReset(Axis := ax); 

mcPower(
	Axis:= ax, 
	Enable:= bAxPower, 
	Enable_Positive:= bAxPower, 
	Enable_Negative:= bAxPower, 
	Override:= 100);

	
mcHome(
	Axis:= ax, 
	Execute:= , 
	Position:= , 
	HomingMode:= , 
	BufferMode:= , 
	Options:= , 
	bCalibrationCam:= NOT(bEndschalter), 
	Done=> homeDone, 
	Busy=> , 
	Active=> , 
	CommandAborted=> , 
	Error=> , 
	ErrorID=> );
	

mcMove(
	Axis:= ax, 
	Execute:= bAxMove, 
	Position:= rPosition, 
	Velocity:= rVel, 
	Acceleration:= 60.0, 
	Deceleration:= 60.0, 
	Jerk:= , 
	BufferMode:= , 
	Options:= , 
	Done=> moveDone, 
	Busy=> , 
	Active=> , 
	CommandAborted=> , 
	Error=> , 
	ErrorID=> );
	
(*
IF NOT benable THEN
	nstate := 0;
END_IF
*)

CASE nstate OF 
	
	0: //off
	estate := eBetriebszustand.off;
	bAxPower := FALSE;
	bAxMove := FALSE;
	
	IF McPower.Status AND benable THEN
		nstate := 20; //Ready
	END_IF
	IF NOT McPower.Status AND bEnable THEN
		nstate:=10;
	END_IF
	
	10: // INIT_Reset
	estate := eBetriebszustand.init;
	mcReset.Execute := TRUE;
	bAxPower:= FALSE;
	bAxMove:= FALSE;
	
	IF McReset.Done THEN
		nstate:= 11; //INIT-Power
	END_IF
	
	11: //INIT-Power
	estate := eBetriebszustand.init;
	bAxPower := TRUE;
	bAxMove := FALSE;
	
	IF Mcpower.Status THEN
		nstate := 20; //Ready
	END_IF
	
	20: //Homing
	estate := eBetriebszustand.init;
	mcHome.Execute := TRUE;
	bAxMove := FALSE;
	
    IF homeDone THEN
      nState := 30;  
    END_IF
	
	30: //Ready
	estate:= eBetriebszustand.ready;
	bAxMove := FALSE;
	
	IF bexecute THEN
		nstate := 40; // Homing
	END_IF
	
	40: //Move
	estate := eBetriebszustand.production;
	bAxMove := TRUE;

	IF moveDone THEN
		nstate := 50; //Done
	END_IF

	50: //Done
	estate := eBetriebszustand.done;
	bAxMove := FALSE;
	
	IF NOT bexecute THEN
		nstate := 20; // Ready
	END_IF
	
END_CASE

END_FUNCTION_BLOCK

// ---- POUs/Manipulator/FB_Robotsteuerung.TcPOU
FUNCTION_BLOCK FB_Robotsteuerung
VAR_INPUT
	bEnable   : BOOL;
  	bExecute  : BOOL;
	bxposition : REAL;
	byposition : REAL;
	bzposition : REAL;
	
	bxEndschalter: BOOL;
	byEndschalter: BOOL;
	bzEndschalter: BOOL;
	bGEndschalter: BOOL;
	
	
END_VAR
VAR_OUTPUT
	estate : eBetriebszustand;
	movedone : BOOL;
END_VAR
VAR
	fbXAchse : FB_Manachse;
	fbYAchse : FB_Manachse;
	fbZAchse : FB_Manachse;
	fbGAchse : FB_ManAchse;  
	nstate : INT := 0;
	currentpos : REAL;
	
	
END_VAR
VAR_IN_OUT
    // Achsen-Referenzen 
    ax_ManX    : AXIS_REF;   
    ax_ManY    : AXIS_REF;   
    ax_ManZ    : AXIS_REF;  
	ax_ManG    : AXIS_REF;   
END_VAR

fbXAchse(
	benable:= , 
	bexecute:= , 
	bEndschalter:= bxEndschalter, 
	rPosition:= bxposition, 
	rVel:= 30, 
	estate=> , 
	ax:= ax_ManX);
	
fbYAchse(
	benable:= , 
	bexecute:= , 
	bEndschalter:= bxEndschalter, 
	rPosition:= byposition, 
	rVel:= 30, 
	estate=> , 
	ax:= ax_ManY);
	
fbZAchse(
	benable:= , 
	bexecute:= , 
	bEndschalter:= bzEndschalter, 
	rPosition:= bzposition, 
	rVel:= 30, 
	estate=> , 
	ax:= ax_ManZ );
	
fbGAchse(
	benable:= , 
	bexecute:= , 
	bEndschalter:= bGEndschalter, 
	rPosition:= , 
	rVel:= 10, 
	estate=> , 
	ax:= ax_ManG);
	
	
CASE nstate OF
	0: //off
	estate := eBetriebszustand.off;
	fbxAchse.benable := FALSE;
	fbyAchse.benable := FALSE;
	fbzAchse.benable := FALSE;
	fbGAchse.benable := FALSE;
	
	IF bEnable THEN
		nstate := 10;
	END_IF
	
	10: //INIT
	fbxAchse.benable := TRUE;
	fbyAchse.benable := TRUE;
	fbzAchse.benable := TRUE;
	fbGAchse.benable := TRUE;
	
	IF fbxAchse.estate = eBetriebszustand.ready AND 
		fbyAchse.estate = eBetriebszustand.ready AND
		fbzAchse.estate = eBetriebszustand.ready THEN
		nstate := 20;
		currentpos := 0.0;
	END_IF
	
	20: // Ready
	eState := eBetriebszustand.ready;
	fbxAchse.benable := TRUE;
	fbyAchse.benable := TRUE;
	fbzAchse.benable := TRUE;
	fbGAchse.benable := TRUE;
	
	IF bexecute AND currentpos < 50.0 THEN
		nstate := 30;
	ELSIF bexecute AND currentpos > 50.0 THEN
		nstate := 60;
	END_IF
	
	30: // MOVEXY
	eState := eBetriebszustand.production;
	fbXAchse.bexecute := TRUE;
	fbYAchse.bexecute := TRUE;
	
	IF fbXAchse.estate = eBetriebszustand.done AND 
		fbYAchse.estate = eBetriebszustand.done THEN
		fbXAchse.bexecute := FALSE;
		fbYAchse.bexecute := FALSE;
		nstate := 40;
	END_IF
	
	40: //MoveZ
	eState := eBetriebszustand.production;
	fbZAchse.bexecute := TRUE;
	
	IF fbZAchse.estate = eBetriebszustand.done THEN
		currentpos := bzposition;
		fbXAchse.bexecute := FALSE;
		nstate  := 50;
	END_IF
	
	50: //Gripper oeffnen
	eState := eBetriebszustand.production;
	fbGAchse.rPosition := 0;
	fbGAchse.bexecute := TRUE;
	
	IF fbGAchse.estate = eBetriebszustand.done THEN
		fbGAchse.bexecute := FALSE;
		nstate := 100;
	END_IF
	
	60: //Gripper oeffnen
	eState := eBetriebszustand.production;
	fbGAchse.rPosition := 8;
	fbGAchse.bexecute := TRUE;
	
	IF fbGAchse.estate = eBetriebszustand.done THEN
		fbGAchse.bexecute := FALSE;
		nstate := 70;
	END_IF	
	
	70: //MoveZ
	eState := eBetriebszustand.production;
	fbZAchse.bexecute := TRUE;
	
	IF fbZAchse.estate = eBetriebszustand.done THEN
		currentpos := bzposition;
		fbXAchse.bexecute := FALSE;
		nstate  := 100;
	END_IF
	
	100: //done
	eState := eBetriebszustand.done;
	
	IF NOT bexecute THEN
		nstate := 20;
	END_IF
	
END_CASE

END_FUNCTION_BLOCK

// ---- POUs/FB_Manipulatormodul.TcPOU
FUNCTION_BLOCK FB_Manipulatormodul
VAR_INPUT
	bEnable : BOOL;
	bExecute : BOOL;
	
	pXhome : REAL;
	pYhome : REAL;
	pZhome : REAL;
	
	pXconv : REAL;
	pYconv : REAL;
	pZconv : REAL;
	
	pXscale : REAL;
	pYscale : REAL;
	pZscale : REAL;
	
	pXheat : REAL;
	pYheat : REAL;
	pZheat : REAL;
	
	pX1stor : REAL;
	pX2stor : REAL;
	pX3stor : REAL;
	pX4stor : REAL;
	pYstor : REAL;
	pZstor : REAL;
	
	estateE : eBetriebszustand;
	
	bxEndschalter: BOOL;
	byEndschalter: BOOL;
	bzEndschalter: BOOL;
	bGEndschalter: BOOL;
	
END_VAR
VAR_OUTPUT
	estate : eBetriebszustand;
END_VAR
VAR
	fbRobotsteuerung : FB_Robotsteuerung;
	fbTON : TON;
	nstate : INT := 0;
	
	targX   : REAL;
  	targY   : REAL;
 	targZ   : REAL;
  	goRobot : BOOL;
END_VAR
VAR_IN_OUT
    // Achsen-Referenzen 
    ax_ManX    : AXIS_REF;   
    ax_ManY    : AXIS_REF;   
    ax_ManZ    : AXIS_REF;  
	ax_ManG    : AXIS_REF;   
END_VAR

fbRobotsteuerung(
	bEnable:= , 
	bExecute:= goRobot, 
	bxposition:= targX, 
	byposition:= targY, 
	bzposition:= targZ, 
	bxEndschalter:= bxEndschalter, 
	byEndschalter:= byEndschalter, 
	bzEndschalter:= bzEndschalter, 
	bGEndschalter:= bGEndschalter, 
	estate=> , 
	movedone=> , 
	ax_ManX:= ax_ManX, 
	ax_ManY:= ax_ManY, 
	ax_ManZ:= ax_ManZ, 
	ax_ManG:= ax_ManG);
	
	fbTON(IN:= , PT:=T#10S , Q=> , ET=> );
CASE nstate OF 
	0: //off
	estate := eBetriebszustand.off;
	fbRobotsteuerung.bEnable := FALSE;
	
	IF bEnable THEN
		nstate := 10;
	END_IF
	
	10: //Init
	estate := eBetriebszustand.init;
	fbRobotsteuerung.bEnable := TRUE;
	
	IF fbRobotsteuerung.estate = eBetriebszustand.ready THEN
		nstate := 20;
	END_IF
	
	20: //Ready
	estate := eBetriebszustand.ready;
	fbRobotsteuerung.bEnable := TRUE;
	
	IF bExecute THEN
		nState := 30; 
	END_IF
	
	30: //Move to Conveyer
	estate := eBetriebszustand.production;
	targX   := pXconv;
  	targY   := pYconv;
 	targZ   := pZconv;
  	goRobot := TRUE;
	
	IF fbRobotsteuerung.estate = eBetriebszustand.done AND
		estateE = eBetriebszustand.done THEN
		goRobot := FALSE;
		nstate := 40;
	END_IF
	
	40: //Lift Z Achse
	estate := eBetriebszustand.production;
	targX   := pXconv;
  	targY   := pYconv;
 	targZ   := pZhome;
  	goRobot := TRUE;


	IF fbRobotsteuerung.estate = eBetriebszustand.done THEN
		goRobot := FALSE;
		nstate := 50;
	END_IF
	
	50: //scale
	estate := eBetriebszustand.production;
	targX   := pXscale;
  	targY   := pYscale;
 	targZ   := pZscale;
  	goRobot := TRUE;
	fbTON.IN := TRUE;

	IF fbRobotsteuerung.estate = eBetriebszustand.done AND
		fbTON.Q = TRUE THEN
		fbTON.IN := FALSE;
		goRobot := FALSE;
		nstate := 60;
	END_IF
	
	60: //Lift Z Achse
	estate := eBetriebszustand.production;
	targX   := pXscale;
  	targY   := pYscale;
 	targZ   := pZhome;
  	goRobot := TRUE;

	IF fbRobotsteuerung.estate = eBetriebszustand.done THEN
		goRobot := FALSE;
		nstate := 70;
	END_IF
	
	70: //heat
	estate := eBetriebszustand.production;
	targX   := pXheat;
  	targY   := pYheat;
 	targZ   := pZheat;
  	goRobot := TRUE;
	fbTON.IN := TRUE;
	
	IF fbRobotsteuerung.estate = eBetriebszustand.done AND
		fbTON.Q = TRUE THEN
		fbTON.IN := FALSE;
		goRobot := FALSE;
		nstate := 80;
	END_IF

	80: //Lift Z Achse
	estate := eBetriebszustand.production;
	targX   := pXheat;
  	targY   := pYheat;
 	targZ   := pZhome;
  	goRobot := TRUE;

	IF fbRobotsteuerung.estate = eBetriebszustand.done THEN
		goRobot := FALSE;
		nstate := 90;
	END_IF
	
	90: //storage
	estate := eBetriebszustand.production;
	targX   := pX1stor;
  	targY   := pYstor;
 	targZ   := pZstor;
  	goRobot := TRUE;
	fbTON.IN := TRUE;

	IF fbRobotsteuerung.estate = eBetriebszustand.done AND
		fbTON.Q = TRUE THEN
		fbTON.IN := FALSE;
		goRobot := FALSE;
		nstate := 100;
	END_IF
	
	100: //Lift Z Achse
	estate := eBetriebszustand.production;
	targX   := pX1stor;
  	targY   := pYstor;
 	targZ   := pZhome;
  	goRobot := TRUE;

	IF fbRobotsteuerung.estate = eBetriebszustand.done THEN
		goRobot := FALSE;
		nstate := 110;
	END_IF
	
	110: //Home
	estate := eBetriebszustand.production;
	targX   := pXhome;
  	targY   := pYhome;
 	targZ   := pZhome;
  	goRobot := TRUE;

	IF fbRobotsteuerung.estate = eBetriebszustand.done THEN
		goRobot := FALSE;
		nstate := 120;
	END_IF
	
	120: // Done
	estate:= eBetriebszustand.done;
	fbRobotsteuerung.bExecute := FALSE;
	
	
END_CASE

END_FUNCTION_BLOCK

// ---- POUs/FUN_SCALE.TcPOU
FUNCTION FUN_SCALE : REAL
VAR_INPUT
	ix : REAL;
	ixmax : REAL;
	ixmin : REAL;
	rymax : REAL;
	rymin : REAL;
END_VAR
VAR
	rk : REAL := 0;
	rd : REAL := 0;
END_VAR

rk := (rymax - rymin)/(ixmax - ixmin);
rd := rymin - rk * ixmin;

FUN_SCALE := rk * ix + rd;

IF FUN_SCALE > rymax THEN
	FUN_SCALE := rymax;
ELSIF FUN_SCALE < rymin THEN
	FUN_SCALE := rymin;
END_IF

END_FUNCTION

// ---- POUs/FB_Maschinentuer.TcPOU
FUNCTION_BLOCK FB_Maschinentuer
VAR_INPUT
	// Sensor Eingang
	bDoorC : BOOL;
	bDoorO : BOOL;
	// Steuereingänge
	benable :BOOL; //Freigabe für Maschinenstezr
	bOpen : BOOL;
	bClose : BOOL;
END_VAR
VAR_OUTPUT
	// Aktor Ausgang
	bVentil : BOOL;
	// Zustände 
	bError : BOOL;
END_VAR
VAR
	nState : INT := 0;
END_VAR

CASE nstate OF
	0: // Tür geschlosen
		//Ausgänge setzen
		bVentil := TRUE;
		
		//Übergangsbedingung
		IF NOT bDoorc  AND benable THEN
			nstate := 3; // Tür schliesßen
		ELSIF bOpen THEN
			nstate := 1; // Tür öffnen
		END_IF
		
	1: // Tür öffnen
		// Ausgänge setzen
		bVentil := FALSE;
		
		//Übergangsbedingung
		IF bdooro THEN
			nstate := nstate + 1; // Tür geöffnet
		END_IF
		
	2: // Tür geöffnet
		bVentil := FALSE;
		
		IF bclose AND benable THEN
			nstate := 3; //Tür schließen
		END_IF
		
	3: //Tür schliesßen
		bVentil := TRUE;
		
		IF bdoorc THEN
			nstate := 0; //Tür geschlossen
		END_IF
		
END_CASE

END_FUNCTION_BLOCK

// ---- POUs/FB_TEST.TcPOU
FUNCTION_BLOCK FB_TEST
VAR_INPUT
	bVentil : BOOL;
END_VAR
VAR_OUTPUT
	bDoorc : BOOL;
	bDooro : BOOL;
END_VAR
VAR
END_VAR

IF bVentil := FALSE
	//animation.delay (500);
	bDooro := TRUE;
END_IF

IF bVentil := TRUE
	//animation.delay (500);
	bDoorc := FALSE;
END_IF

END_FUNCTION_BLOCK
